FUNCTION_BLOCK FB_PH_Grid_Visu EXTENDS FB_VisuSelector
VAR_INPUT
END_VAR
VAR_OUTPUT
END_VAR
VAR_IN_OUT
  sI_Ary_Fb :   ARRAY[*] OF FB_PH_Grid;
END_VAR
VAR
  pL_Elem_Fb    : POINTER TO FB_PH_Grid;
END_VAR

(*checks*)
IF (ADR(sI_Ary_Fb) = 0) THEN
  F_Report_Error(Report_Error_0Pointer);
  RETURN;
END_IF

(*init fb*)
IF NOT bL_Init THEN
  SUPER^.setAryBounds(iLowerBoundary:=LOWER_BOUND(sI_Ary_Fb, 1), iUpperBoundary:=UPPER_BOUND(sI_Ary_Fb, 1));  
END_IF

(*call*)
SUPER^();
pL_Elem_Fb  := ADR(sI_Ary_Fb[pSelect^]);

END_FUNCTION_BLOCK

(* stored: Version 1.1.0.1, ProductVersion 3.1.4024.3
   POU FB_PH_Grid_Visu: Id {dc6b5099-4caa-44b5-94b6-de2f1612d448}, SpecialFunc None *)
